Staubli VAL3: Day8.dtx

string sInput
lists lResult
  [0]
    string sString
lists lResultSplit
  [0]
    string sString
